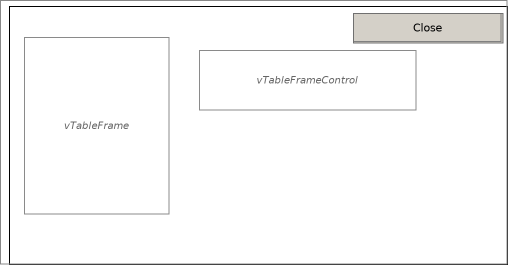
VISUALIZATION vTableFrameDialog  // 508x265
VAR_IN_OUT
	fbTableControl:FB_TableControl;
END_VAR
    Rectangle (9,6 499x259)
    Button (353,13 150x30), "Close"
        OnMouseDown: execute { fbTableControl.stHMI.iDialogNumber:=0; }
    Frame (24,37 145x177)
        shows vTableFrame(fbTablePlace := fbTableControl.arrPlaces[fbTableControl.stHMI.iDialogNumber], fbTableControl := fbTableControl)
    Frame (199,50 217x60)
        shows vTableFrameControl(fbTablePlace := fbTableControl.arrPlaces[fbTableControl.stHMI.iDialogNumber])
END_VISUALIZATION

(* stored: Version 1.1.0.1, ProductVersion 3.1.4024.15
   Visu vTableFrameDialog: Id {28e5882f-fa08-4a56-8b62-21aab374e94f} *)
